{attribute 'qualified_only'}
{attribute 'strict'}
TYPE E_PixelFormat :
(
	RRGGBBAA,
	AARRGGBB,
	xxRRGGBB
);
END_TYPE

(* stored: Version 1.1.0.1, ProductVersion 3.1.4024.15
   DUT E_PixelFormat: Id {418cf84c-0cea-08bb-10b7-e7b0dd213330} *)
